FUNCTION_BLOCK FB_HE_SATT_FilterToTransmission_Test EXTENDS FB_TestSuite


GivenFilterExpectCorrectTransmission();


METHOD PRIVATE GivenFilterExpectCorrectTransmission
VAR
    
END_VAR

TEST('GivenFilterExpectCorrectTransmission');



TEST_FINISHED();
END_METHOD

END_FUNCTION_BLOCK

(* stored: Version 1.1.0.1
   POU FB_HE_SATT_FilterToTransmission_Test: Id {eeaad0ba-8c82-43ea-ad82-ea5fbc896027}, SpecialFunc None
   Method GivenFilterExpectCorrectTransmission: Id {5183906e-5d89-4e8f-ae4b-bfd27aeb0bf5} *)
